FUNCTION CalculateSine : REAL
VAR_INPUT
	angle_in_radians : REAL;
END_VAR

VAR_OUTPUT
	sine_value : REAL;
END_VAR

sine_value := SIN(angle_in_radians);

END_FUNCTION

(* stored: Version 1.1.0.1, ProductVersion 3.1.4024.13
   POU CalculateSine: Id {448da375-44f6-4116-a111-80de455fbe46}, SpecialFunc None *)
